FUNCTION_BLOCK FB_OPCUA_GetRecipe
VAR_INPUT
END_VAR
VAR_OUTPUT
END_VAR
VAR
END_VAR

END_FUNCTION_BLOCK

(* stored: Version 1.1.0.1, ProductVersion 3.1.4024.2
   POU FB_OPCUA_GetRecipe: Id {b1ef5857-878b-4c27-b000-1c88dc25d3c5}, SpecialFunc None *)
